FUNCTION_BLOCK FB_Scheduler_F38
      VAR_INPUT
          currH : WORD;
          currM : WORD;
          currD : WORD;
      END_VAR
      VAR_IN_OUT
          FB_Bacnet : FB_BACnet_DAIKIN_MasterStation_III_No_9;
      END_VAR
      VAR
          i : INT;
          bUnitTriggered : BOOL := FALSE; // New flag to track execution
          prevMinute : WORD := 0;        // New variable to track the previous minute
      END_VAR
      VAR PERSISTENT
          //scheduler var
          bEnSchedF38_ : BOOL := FALSE;
          wSchedWDHourStartF38_ : WORD; 
          wSchedWDMinStartF38_ : WORD; 
          wSchedWEHourStartF38_ : WORD; 
          wSchedWEMinStartF38_ : WORD;
          wSchedWDHourEndF38_ : WORD;
          wSchedWDMinEndF38_ : WORD;
          wSchedWEHourEndF38_ : WORD;
          wSchedWEMinEndF38_ : WORD;
          //unit var
          bUnitF38_ : ARRAY [1..25] OF BOOL;
      END_VAR


        // Reset trigger flag at minute change or at the exact scheduled time
        IF currM <> prevMinute OR 
           (currH = wSchedWDHourStartF38_ AND currM = wSchedWDMinStartF38_) OR 
           (currH = wSchedWDHourEndF38_ AND currM = wSchedWDMinEndF38_) THEN
            bUnitTriggered := FALSE;
            prevMinute := currM;
        END_IF

        // Unit Schedule Enable
        IF bEnSchedF38_ THEN
            // Weekday schedule
            IF currD >= 1 AND currD <= 5 THEN
                IF (wSchedWDHourStartF38_ <> wSchedWDHourEndF38_ OR wSchedWDMinStartF38_ <> wSchedWDMinEndF38_) THEN
                    // Schedule Unit ON
                    IF wSchedWDHourStartF38_ = currH AND wSchedWDMinStartF38_ = currM AND NOT bUnitTriggered THEN
                        bUnitTriggered := TRUE;
                        FOR i := 1 TO 25 DO
                            // Send command unit ON
                            IF bUnitF38_[i] THEN 
                                CASE i OF
                                    1: 
                                        
                                        FB_Bacnet.StartStopCommand_128.bEnWrite := TRUE;
                                        FB_Bacnet.StartStopCommand_128.bVal := TRUE;
                                    2: 
                                        
                                        FB_Bacnet.StartStopCommand_129.bEnWrite := TRUE;
                                        FB_Bacnet.StartStopCommand_129.bVal := TRUE;
                                    3: 
                                        
                                        FB_Bacnet.StartStopCommand_130.bEnWrite := TRUE;
                                        FB_Bacnet.StartStopCommand_130.bVal := TRUE;
                                    4: 
                                        
                                        FB_Bacnet.StartStopCommand_131.bEnWrite := TRUE;
                                        FB_Bacnet.StartStopCommand_131.bVal := TRUE;
                                    5: 
                                        
                                        FB_Bacnet.StartStopCommand_132.bEnWrite := TRUE;
                                        FB_Bacnet.StartStopCommand_132.bVal := TRUE;
                                    6: 
                                        
                                        FB_Bacnet.StartStopCommand_133.bEnWrite := TRUE;
                                        FB_Bacnet.StartStopCommand_133.bVal := TRUE;
                                    7: 
                                        
                                        FB_Bacnet.StartStopCommand_134.bEnWrite := TRUE;
                                        FB_Bacnet.StartStopCommand_134.bVal := TRUE;
                                    8: 
                                        
                                        FB_Bacnet.StartStopCommand_135.bEnWrite := TRUE;
                                        FB_Bacnet.StartStopCommand_135.bVal := TRUE;
                                    9: 
                                        
                                        FB_Bacnet.StartStopCommand_136.bEnWrite := TRUE;
                                        FB_Bacnet.StartStopCommand_136.bVal := TRUE;
                                    10: 
                                        
                                        FB_Bacnet.StartStopCommand_137.bEnWrite := TRUE;
                                        FB_Bacnet.StartStopCommand_137.bVal := TRUE;
                                    11: 
                                        
                                        FB_Bacnet.StartStopCommand_138.bEnWrite := TRUE;
                                        FB_Bacnet.StartStopCommand_138.bVal := TRUE;
                                    12: 
                                        
                                        FB_Bacnet.StartStopCommand_139.bEnWrite := TRUE;
                                        FB_Bacnet.StartStopCommand_139.bVal := TRUE;
                                    13: 
                                        
                                        FB_Bacnet.StartStopCommand_140.bEnWrite := TRUE;
                                        FB_Bacnet.StartStopCommand_140.bVal := TRUE;
                                    14: 
                                        
                                        FB_Bacnet.StartStopCommand_141.bEnWrite := TRUE;
                                        FB_Bacnet.StartStopCommand_141.bVal := TRUE;
                                    15: 
                                        
                                        FB_Bacnet.StartStopCommand_142.bEnWrite := TRUE;
                                        FB_Bacnet.StartStopCommand_142.bVal := TRUE;
                                    16: 
                                        
                                        FB_Bacnet.StartStopCommand_143.bEnWrite := TRUE;
                                        FB_Bacnet.StartStopCommand_143.bVal := TRUE;
                                    17: 
                                        
                                        FB_Bacnet.StartStopCommand_144.bEnWrite := TRUE;
                                        FB_Bacnet.StartStopCommand_144.bVal := TRUE;
                                    18: 
                                        
                                        FB_Bacnet.StartStopCommand_145.bEnWrite := TRUE;
                                        FB_Bacnet.StartStopCommand_145.bVal := TRUE;
                                    19: 
                                        
                                        FB_Bacnet.StartStopCommand_146.bEnWrite := TRUE;
                                        FB_Bacnet.StartStopCommand_146.bVal := TRUE;
                                    20: 
                                        
                                        FB_Bacnet.StartStopCommand_147.bEnWrite := TRUE;
                                        FB_Bacnet.StartStopCommand_147.bVal := TRUE;
                                    21: 
                                        
                                        FB_Bacnet.StartStopCommand_148.bEnWrite := TRUE;
                                        FB_Bacnet.StartStopCommand_148.bVal := TRUE;
                                    22: 
                                        
                                        FB_Bacnet.StartStopCommand_149.bEnWrite := TRUE;
                                        FB_Bacnet.StartStopCommand_149.bVal := TRUE;
                                    23: 
                                        
                                        FB_Bacnet.StartStopCommand_176.bEnWrite := TRUE;
                                        FB_Bacnet.StartStopCommand_176.bVal := TRUE;
                                    24: 
                                        
                                        FB_Bacnet.StartStopCommand_241.bEnWrite := TRUE;
                                        FB_Bacnet.StartStopCommand_241.bVal := TRUE;
                                    25: 
                                        
                                        FB_Bacnet.StartStopCommand_226.bEnWrite := TRUE;
                                        FB_Bacnet.StartStopCommand_226.bVal := TRUE;
                                END_CASE
                            END_IF
                        END_FOR
                    END_IF
                    // Schedule Unit OFF
                    IF wSchedWDHourEndF38_ = currH AND wSchedWDMinEndF38_ = currM AND NOT bUnitTriggered THEN
                        bUnitTriggered := TRUE;
                        FOR i := 1 TO 25 DO
                            // Send command unit OFF
                            IF bUnitF38_[i] THEN 
                                CASE i OF
                                    1: 
                                        
                                        FB_Bacnet.StartStopCommand_128.bEnWrite := TRUE;
                                        FB_Bacnet.StartStopCommand_128.bVal := FALSE;
                                    2: 
                                        
                                        FB_Bacnet.StartStopCommand_129.bEnWrite := TRUE;
                                        FB_Bacnet.StartStopCommand_129.bVal := FALSE;
                                    3: 
                                        
                                        FB_Bacnet.StartStopCommand_130.bEnWrite := TRUE;
                                        FB_Bacnet.StartStopCommand_130.bVal := FALSE;
                                    4: 
                                        
                                        FB_Bacnet.StartStopCommand_131.bEnWrite := TRUE;
                                        FB_Bacnet.StartStopCommand_131.bVal := FALSE;
                                    5: 
                                        
                                        FB_Bacnet.StartStopCommand_132.bEnWrite := TRUE;
                                        FB_Bacnet.StartStopCommand_132.bVal := FALSE;
                                    6: 
                                        
                                        FB_Bacnet.StartStopCommand_133.bEnWrite := TRUE;
                                        FB_Bacnet.StartStopCommand_133.bVal := FALSE;
                                    7: 
                                        
                                        FB_Bacnet.StartStopCommand_134.bEnWrite := TRUE;
                                        FB_Bacnet.StartStopCommand_134.bVal := FALSE;
                                    8: 
                                        
                                        FB_Bacnet.StartStopCommand_135.bEnWrite := TRUE;
                                        FB_Bacnet.StartStopCommand_135.bVal := FALSE;
                                    9: 
                                        
                                        FB_Bacnet.StartStopCommand_136.bEnWrite := TRUE;
                                        FB_Bacnet.StartStopCommand_136.bVal := FALSE;
                                    10: 
                                        
                                        FB_Bacnet.StartStopCommand_137.bEnWrite := TRUE;
                                        FB_Bacnet.StartStopCommand_137.bVal := FALSE;
                                    11: 
                                        
                                        FB_Bacnet.StartStopCommand_138.bEnWrite := TRUE;
                                        FB_Bacnet.StartStopCommand_138.bVal := FALSE;
                                    12: 
                                        
                                        FB_Bacnet.StartStopCommand_139.bEnWrite := TRUE;
                                        FB_Bacnet.StartStopCommand_139.bVal := FALSE;
                                    13: 
                                        
                                        FB_Bacnet.StartStopCommand_140.bEnWrite := TRUE;
                                        FB_Bacnet.StartStopCommand_140.bVal := FALSE;
                                    14: 
                                        
                                        FB_Bacnet.StartStopCommand_141.bEnWrite := TRUE;
                                        FB_Bacnet.StartStopCommand_141.bVal := FALSE;
                                    15: 
                                        
                                        FB_Bacnet.StartStopCommand_142.bEnWrite := TRUE;
                                        FB_Bacnet.StartStopCommand_142.bVal := FALSE;
                                    16: 
                                        
                                        FB_Bacnet.StartStopCommand_143.bEnWrite := TRUE;
                                        FB_Bacnet.StartStopCommand_143.bVal := FALSE;
                                    17: 
                                        
                                        FB_Bacnet.StartStopCommand_144.bEnWrite := TRUE;
                                        FB_Bacnet.StartStopCommand_144.bVal := FALSE;
                                    18: 
                                        
                                        FB_Bacnet.StartStopCommand_145.bEnWrite := TRUE;
                                        FB_Bacnet.StartStopCommand_145.bVal := FALSE;
                                    19: 
                                        
                                        FB_Bacnet.StartStopCommand_146.bEnWrite := TRUE;
                                        FB_Bacnet.StartStopCommand_146.bVal := FALSE;
                                    20: 
                                        
                                        FB_Bacnet.StartStopCommand_147.bEnWrite := TRUE;
                                        FB_Bacnet.StartStopCommand_147.bVal := FALSE;
                                    21: 
                                        
                                        FB_Bacnet.StartStopCommand_148.bEnWrite := TRUE;
                                        FB_Bacnet.StartStopCommand_148.bVal := FALSE;
                                    22: 
                                        
                                        FB_Bacnet.StartStopCommand_149.bEnWrite := TRUE;
                                        FB_Bacnet.StartStopCommand_149.bVal := FALSE;
                                    23: 
                                        
                                        FB_Bacnet.StartStopCommand_176.bEnWrite := TRUE;
                                        FB_Bacnet.StartStopCommand_176.bVal := FALSE;
                                    24: 
                                        
                                        FB_Bacnet.StartStopCommand_241.bEnWrite := TRUE;
                                        FB_Bacnet.StartStopCommand_241.bVal := FALSE;
                                    25: 
                                        
                                        FB_Bacnet.StartStopCommand_226.bEnWrite := TRUE;
                                        FB_Bacnet.StartStopCommand_226.bVal := FALSE;
                                END_CASE
                            END_IF
                        END_FOR
                    END_IF
                END_IF
            END_IF
        END_IF

        // Weekend schedule
        IF currD = 0 OR currD = 6 THEN
            IF (wSchedWEHourStartF38_ <> wSchedWEHourEndF38_ OR wSchedWEMinStartF38_ <> wSchedWEMinEndF38_) THEN
                // Schedule Unit ON
                IF wSchedWEHourStartF38_ = currH AND wSchedWEMinStartF38_ = currM AND NOT bUnitTriggered THEN
                    bUnitTriggered := TRUE;
                    FOR i := 1 TO 25 DO
                        // Send command unit ON
                        IF bUnitF38_[i] THEN 
                            CASE i OF
                                1: 
                                    
                                    FB_Bacnet.StartStopCommand_128.bEnWrite := TRUE;
                                    FB_Bacnet.StartStopCommand_128.bVal := TRUE;
                                2: 
                                    
                                    FB_Bacnet.StartStopCommand_129.bEnWrite := TRUE;
                                    FB_Bacnet.StartStopCommand_129.bVal := TRUE;
                                3: 
                                    
                                    FB_Bacnet.StartStopCommand_130.bEnWrite := TRUE;
                                    FB_Bacnet.StartStopCommand_130.bVal := TRUE;
                                4: 
                                    
                                    FB_Bacnet.StartStopCommand_131.bEnWrite := TRUE;
                                    FB_Bacnet.StartStopCommand_131.bVal := TRUE;
                                5: 
                                    
                                    FB_Bacnet.StartStopCommand_132.bEnWrite := TRUE;
                                    FB_Bacnet.StartStopCommand_132.bVal := TRUE;
                                6: 
                                    
                                    FB_Bacnet.StartStopCommand_133.bEnWrite := TRUE;
                                    FB_Bacnet.StartStopCommand_133.bVal := TRUE;
                                7: 
                                    
                                    FB_Bacnet.StartStopCommand_134.bEnWrite := TRUE;
                                    FB_Bacnet.StartStopCommand_134.bVal := TRUE;
                                8: 
                                    
                                    FB_Bacnet.StartStopCommand_135.bEnWrite := TRUE;
                                    FB_Bacnet.StartStopCommand_135.bVal := TRUE;
                                9: 
                                    
                                    FB_Bacnet.StartStopCommand_136.bEnWrite := TRUE;
                                    FB_Bacnet.StartStopCommand_136.bVal := TRUE;
                                10: 
                                    
                                    FB_Bacnet.StartStopCommand_137.bEnWrite := TRUE;
                                    FB_Bacnet.StartStopCommand_137.bVal := TRUE;
                                11: 
                                    
                                    FB_Bacnet.StartStopCommand_138.bEnWrite := TRUE;
                                    FB_Bacnet.StartStopCommand_138.bVal := TRUE;
                                12: 
                                    
                                    FB_Bacnet.StartStopCommand_139.bEnWrite := TRUE;
                                    FB_Bacnet.StartStopCommand_139.bVal := TRUE;
                                13: 
                                    
                                    FB_Bacnet.StartStopCommand_140.bEnWrite := TRUE;
                                    FB_Bacnet.StartStopCommand_140.bVal := TRUE;
                                14: 
                                    
                                    FB_Bacnet.StartStopCommand_141.bEnWrite := TRUE;
                                    FB_Bacnet.StartStopCommand_141.bVal := TRUE;
                                15: 
                                    
                                    FB_Bacnet.StartStopCommand_142.bEnWrite := TRUE;
                                    FB_Bacnet.StartStopCommand_142.bVal := TRUE;
                                16: 
                                    
                                    FB_Bacnet.StartStopCommand_143.bEnWrite := TRUE;
                                    FB_Bacnet.StartStopCommand_143.bVal := TRUE;
                                17: 
                                    
                                    FB_Bacnet.StartStopCommand_144.bEnWrite := TRUE;
                                    FB_Bacnet.StartStopCommand_144.bVal := TRUE;
                                18: 
                                    
                                    FB_Bacnet.StartStopCommand_145.bEnWrite := TRUE;
                                    FB_Bacnet.StartStopCommand_145.bVal := TRUE;
                                19: 
                                    
                                    FB_Bacnet.StartStopCommand_146.bEnWrite := TRUE;
                                    FB_Bacnet.StartStopCommand_146.bVal := TRUE;
                                20: 
                                    
                                    FB_Bacnet.StartStopCommand_147.bEnWrite := TRUE;
                                    FB_Bacnet.StartStopCommand_147.bVal := TRUE;
                                21: 
                                    
                                    FB_Bacnet.StartStopCommand_148.bEnWrite := TRUE;
                                    FB_Bacnet.StartStopCommand_148.bVal := TRUE;
                                22: 
                                    
                                    FB_Bacnet.StartStopCommand_149.bEnWrite := TRUE;
                                    FB_Bacnet.StartStopCommand_149.bVal := TRUE;
                                23: 
                                    
                                    FB_Bacnet.StartStopCommand_176.bEnWrite := TRUE;
                                    FB_Bacnet.StartStopCommand_176.bVal := TRUE;
                                24: 
                                    
                                    FB_Bacnet.StartStopCommand_241.bEnWrite := TRUE;
                                    FB_Bacnet.StartStopCommand_241.bVal := TRUE;
                                25: 
                                    
                                    FB_Bacnet.StartStopCommand_226.bEnWrite := TRUE;
                                    FB_Bacnet.StartStopCommand_226.bVal := TRUE;
                            END_CASE
                        END_IF
                    END_FOR        
                END_IF
                // Schedule Unit OFF
                IF wSchedWEHourEndF38_ = currH AND wSchedWEMinEndF38_ = currM AND NOT bUnitTriggered THEN
                    bUnitTriggered := TRUE;
                    FOR i := 1 TO 25 DO
                        // Send command unit OFF
                        IF bUnitF38_[i] THEN 
                            CASE i OF
                                1: 
                                    
                                    FB_Bacnet.StartStopCommand_128.bEnWrite := TRUE;
                                    FB_Bacnet.StartStopCommand_128.bVal := FALSE;
                                2: 
                                    
                                    FB_Bacnet.StartStopCommand_129.bEnWrite := TRUE;
                                    FB_Bacnet.StartStopCommand_129.bVal := FALSE;
                                3: 
                                    
                                    FB_Bacnet.StartStopCommand_130.bEnWrite := TRUE;
                                    FB_Bacnet.StartStopCommand_130.bVal := FALSE;
                                4: 
                                    
                                    FB_Bacnet.StartStopCommand_131.bEnWrite := TRUE;
                                    FB_Bacnet.StartStopCommand_131.bVal := FALSE;
                                5: 
                                    
                                    FB_Bacnet.StartStopCommand_132.bEnWrite := TRUE;
                                    FB_Bacnet.StartStopCommand_132.bVal := FALSE;
                                6: 
                                    
                                    FB_Bacnet.StartStopCommand_133.bEnWrite := TRUE;
                                    FB_Bacnet.StartStopCommand_133.bVal := FALSE;
                                7: 
                                    
                                    FB_Bacnet.StartStopCommand_134.bEnWrite := TRUE;
                                    FB_Bacnet.StartStopCommand_134.bVal := FALSE;
                                8: 
                                    
                                    FB_Bacnet.StartStopCommand_135.bEnWrite := TRUE;
                                    FB_Bacnet.StartStopCommand_135.bVal := FALSE;
                                9: 
                                    
                                    FB_Bacnet.StartStopCommand_136.bEnWrite := TRUE;
                                    FB_Bacnet.StartStopCommand_136.bVal := FALSE;
                                10: 
                                    
                                    FB_Bacnet.StartStopCommand_137.bEnWrite := TRUE;
                                    FB_Bacnet.StartStopCommand_137.bVal := FALSE;
                                11: 
                                    
                                    FB_Bacnet.StartStopCommand_138.bEnWrite := TRUE;
                                    FB_Bacnet.StartStopCommand_138.bVal := FALSE;
                                12: 
                                    
                                    FB_Bacnet.StartStopCommand_139.bEnWrite := TRUE;
                                    FB_Bacnet.StartStopCommand_139.bVal := FALSE;
                                13: 
                                    
                                    FB_Bacnet.StartStopCommand_140.bEnWrite := TRUE;
                                    FB_Bacnet.StartStopCommand_140.bVal := FALSE;
                                14: 
                                    
                                    FB_Bacnet.StartStopCommand_141.bEnWrite := TRUE;
                                    FB_Bacnet.StartStopCommand_141.bVal := FALSE;
                                15: 
                                    
                                    FB_Bacnet.StartStopCommand_142.bEnWrite := TRUE;
                                    FB_Bacnet.StartStopCommand_142.bVal := FALSE;
                                16: 
                                    
                                    FB_Bacnet.StartStopCommand_143.bEnWrite := TRUE;
                                    FB_Bacnet.StartStopCommand_143.bVal := FALSE;
                                17: 
                                    
                                    FB_Bacnet.StartStopCommand_144.bEnWrite := TRUE;
                                    FB_Bacnet.StartStopCommand_144.bVal := FALSE;
                                18: 
                                    
                                    FB_Bacnet.StartStopCommand_145.bEnWrite := TRUE;
                                    FB_Bacnet.StartStopCommand_145.bVal := FALSE;
                                19: 
                                    
                                    FB_Bacnet.StartStopCommand_146.bEnWrite := TRUE;
                                    FB_Bacnet.StartStopCommand_146.bVal := FALSE;
                                20: 
                                    
                                    FB_Bacnet.StartStopCommand_147.bEnWrite := TRUE;
                                    FB_Bacnet.StartStopCommand_147.bVal := FALSE;
                                21: 
                                    
                                    FB_Bacnet.StartStopCommand_148.bEnWrite := TRUE;
                                    FB_Bacnet.StartStopCommand_148.bVal := FALSE;
                                22: 
                                    
                                    FB_Bacnet.StartStopCommand_149.bEnWrite := TRUE;
                                    FB_Bacnet.StartStopCommand_149.bVal := FALSE;
                                23: 
                                    
                                    FB_Bacnet.StartStopCommand_176.bEnWrite := TRUE;
                                    FB_Bacnet.StartStopCommand_176.bVal := FALSE;
                                24: 
                                    
                                    FB_Bacnet.StartStopCommand_241.bEnWrite := TRUE;
                                    FB_Bacnet.StartStopCommand_241.bVal := FALSE;
                                25: 
                                    
                                    FB_Bacnet.StartStopCommand_226.bEnWrite := TRUE;
                                    FB_Bacnet.StartStopCommand_226.bVal := FALSE;
                            END_CASE
                        END_IF
                    END_FOR
                END_IF
            END_IF
        END_IF

END_FUNCTION_BLOCK

(* stored: Version 1.1.0.1, ProductVersion 3.1.4024.14
   POU FB_Scheduler_F38: Id {08181ac3-5ead-4737-ac4d-656f72650346}, SpecialFunc None *)
